//==================================================================================================
//								RJM Maszyny sp. z o.o.
//									04.02.2022
//	Obsługa elektrozaworu 5/2 bistabilny
// 	v1.0	|| TC v 3.1.4024.22		|| - pierwsza wersja
//==================================================================================================
FUNCTION_BLOCK FB_Elektrozawor_5na2_2Cewki IMPLEMENTS I_Elektrozawor_5na
VAR
	fbCewkaA								: FB_ElektrozaworCewka; //sterowanie wyjscie 2
	fbCewkaB								: FB_ElektrozaworCewka; //sterowanie wyjscie 4
END_VAR

//==================================================================================================
//								RJM Maszyny sp. z o.o.
//									04.02.2022
//	Włączenie cewki - wyjscie 2
// 	v1.0	|| TC v 3.1.4024.22		|| - pierwsza wersja
//==================================================================================================
METHOD WlaczWyjscie2 : BOOL
VAR_INPUT
END_VAR
fbCewkaA.Wlacz ();
END_METHOD

//==================================================================================================
//								RJM Maszyny sp. z o.o.
//									04.02.2022
//	Włączenie cewki - wyjscie 4
// 	v1.0	|| TC v 3.1.4024.22		|| - pierwsza wersja
//==================================================================================================
METHOD WlaczWyjscie4 : BOOL
VAR_INPUT
END_VAR
fbCewkaB.Wlacz ();
END_METHOD

//==================================================================================================
//								RJM Maszyny sp. z o.o.
//									04.02.2022
//	Wyłączenie cewki - wyjscie 2
// 	v1.0	|| TC v 3.1.4024.22		|| - pierwsza wersja
//==================================================================================================METHOD WylaczWyjscie2 : BOOL
VAR_INPUT
END_VAR
fbCewkaA.Wylacz ();
END_METHOD

//==================================================================================================
//								RJM Maszyny sp. z o.o.
//									04.02.2022
//	Wyłączenie cewki - wyjscie 4
// 	v1.0	|| TC v 3.1.4024.22		|| - pierwsza wersja
//==================================================================================================
METHOD WylaczWyjscie4 : BOOL
VAR_INPUT
END_VAR
fbCewkaB.Wylacz ();
END_METHOD

END_FUNCTION_BLOCK

(* stored: Version 1.1.0.1, ProductVersion 3.1.4024.11
   POU FB_Elektrozawor_5na2_2Cewki: Id {3d99ae90-0092-4a28-a425-90fd1fee7a8b}, SpecialFunc None
   Method WlaczWyjscie2: Id {ca2bcd17-18ec-4a83-aa5c-76fdf107ba9a}
   Method WlaczWyjscie4: Id {6d51c73b-5893-4a11-abc8-57d8c746097f}
   Method WylaczWyjscie2: Id {5712b962-e562-463c-9277-2760aecbb3e8}
   Method WylaczWyjscie4: Id {aae23a92-0435-4045-b965-8391db85db8d} *)
